Staubli VAL3: start.pgx

program start()
  local num l_i
  local num l_sum
begin
  //
  call cst:init()
  call chkLife()
  if blifebit
    call init()
    taskCreateSync "T4ms",0.004,bOverrun,Task4ms()
  endIf
end
